FUNCTION F_ComputeFixed32Size : UDINT
VAR_INPUT
    {attribute 'analysis' := '-33' }
    nValue : UDINT;
END_VAR


F_ComputeFixed32Size := GCL_PB.cLittleEndian32Size;

END_FUNCTION

(* stored: Version 1.1.0.1
   POU F_ComputeFixed32Size: Id {766ea878-df40-4de8-81d4-27ffd1dd4c9d}, SpecialFunc None *)
